{attribute 'qualified_only'}
{attribute 'strict'}
TYPE eErrorReadWrite :
(
	eNoError							:= 0,
	eErrorRead							:= 1,
	eErrorWrite							:= 2,
	eErrorSizeFloatValueRead			:= 3,
	eErrorSizeValueWrite				:= 4
);
END_TYPE

(* stored: Version 1.1.0.1, ProductVersion 3.1.4024.6
   DUT eErrorReadWrite: Id {9d52db5c-3abd-4af3-b780-d73fe1d76b98} *)
